PROGRAM MAIN
VAR
END_VAR

END_PROGRAM

(* stored: Version 1.1.0.1
   POU MAIN: Id {3e191fa6-7ea5-48e4-abf7-470effa94126} *)
